# EPICS substitutions: OPCUA/OPCUA-IOC-01App/Db/MAPS_vacuum.substitutions
file "$(TOP)/OPCUA-IOC-01App/Db/MAPS_vacuum_other.template" {
	pattern{ P, R, SUBS, DEBUG, RECORD_TYPE, PV_NAME, NAME_PREFIX, NAME_SUFFIX}

#   General records:
	{ "\$(P)", "\$(R)", "\$(SUBS)", "\$(DEBUG=0)", "stringin", "PE_UNDERRANGE", "\$(NAME_PREFIX)", "Statuses.PE_Underrange_Control" }
    { "\$(P)", "\$(R)", "\$(SUBS)", "\$(DEBUG=0)", "stringin", "UNIT",          "\$(NAME_PREFIX)", "Statuses.Pressure_Unit" }
    { "\$(P)", "\$(R)", "\$(SUBS)", "\$(DEBUG=0)", "stringin", "ERROR",         "\$(NAME_PREFIX)", "Statuses.TPG_Error" }
    { "\$(P)", "\$(R)", "\$(SUBS)", "\$(DEBUG=0)", "bi",       "HEALTHY",       "\$(NAME_PREFIX)", "Statuses.TPG_Healthy" }

#   Channel 1 / Sensor A1:
    { "\$(P)", "\$(R)", "\$(SUBS)", "\$(DEBUG=0)", "stringin", "MEASURED_VALUE_A1",    "\$(NAME_PREFIX)", "Sensor_A1.Measured_Value_Status" }
    { "\$(P)", "\$(R)", "\$(SUBS)", "\$(DEBUG=0)", "stringin", "MEASURING_CIRCUIT_A1", "\$(NAME_PREFIX)", "Sensor_A1.Measuring_Circuit_Status" }
    { "\$(P)", "\$(R)", "\$(SUBS)", "\$(DEBUG=0)", "stringin", "FILTER_TIME_CONST_A1", "\$(NAME_PREFIX)", "Sensor_A1.Filter_Time_Constant" }

#   Relay 1:
    { "\$(P)", "\$(R)", "\$(SUBS)", "\$(DEBUG=0)", "ai",       "THRESHOLD_LOW_A1",      "\$(NAME_PREFIX)", "Relay1.Lower_Threshold" }
    { "\$(P)", "\$(R)", "\$(SUBS)", "\$(DEBUG=0)", "ai",       "THRESHOLD_HI_A1",       "\$(NAME_PREFIX)", "Relay1.Upper_Threshold" }
    { "\$(P)", "\$(R)", "\$(SUBS)", "\$(DEBUG=0)", "stringin", "SWITCH_FUNC_ASSIGN_A1", "\$(NAME_PREFIX)", "Relay1.Switching_Function_Assignment" }
    { "\$(P)", "\$(R)", "\$(SUBS)", "\$(DEBUG=0)", "stringin", "SWITCH_FUNC_STATUS_A1", "\$(NAME_PREFIX)", "Relay1.Switching_Function_Status" }

#   Channel 2 / Sensor A2:
    { "\$(P)", "\$(R)", "\$(SUBS)", "\$(DEBUG=0)", "stringin", "MEASURED_VALUE_A2",    "\$(NAME_PREFIX)", "Sensor_A2.Measured_Value_Status" }
    { "\$(P)", "\$(R)", "\$(SUBS)", "\$(DEBUG=0)", "stringin", "MEASURING_CIRCUIT_A2", "\$(NAME_PREFIX)", "Sensor_A2.Measuring_Circuit_Status" }
    { "\$(P)", "\$(R)", "\$(SUBS)", "\$(DEBUG=0)", "stringin", "FILTER_TIME_CONST_A2", "\$(NAME_PREFIX)", "Sensor_A2.Filter_Time_Constant" }

#   Relay 2:
    { "\$(P)", "\$(R)", "\$(SUBS)", "\$(DEBUG=0)", "ai",       "THRESHOLD_LOW_A2",      "\$(NAME_PREFIX)", "Relay2.Lower_Threshold" }
    { "\$(P)", "\$(R)", "\$(SUBS)", "\$(DEBUG=0)", "ai",       "THRESHOLD_HI_A2",       "\$(NAME_PREFIX)", "Relay2.Upper_Threshold" }
    { "\$(P)", "\$(R)", "\$(SUBS)", "\$(DEBUG=0)", "stringin", "SWITCH_FUNC_ASSIGN_A2", "\$(NAME_PREFIX)", "Relay2.Switching_Function_Assignment" }
    { "\$(P)", "\$(R)", "\$(SUBS)", "\$(DEBUG=0)", "stringin", "SWITCH_FUNC_STATUS_A2", "\$(NAME_PREFIX)", "Relay2.Switching_Function_Status" }

#   Channel 3 / Sensor B1:
    { "\$(P)", "\$(R)", "\$(SUBS)", "\$(DEBUG=0)", "stringin", "MEASURED_VALUE_B1",    "\$(NAME_PREFIX)", "Sensor_B1.Measured_Value_Status" }
    { "\$(P)", "\$(R)", "\$(SUBS)", "\$(DEBUG=0)", "stringin", "MEASURING_CIRCUIT_B1", "\$(NAME_PREFIX)", "Sensor_B1.Measuring_Circuit_Status" }
    { "\$(P)", "\$(R)", "\$(SUBS)", "\$(DEBUG=0)", "stringin", "FILTER_TIME_CONST_B1", "\$(NAME_PREFIX)", "Sensor_B1.Filter_Time_Constant" }

#   Relay 3:
    { "\$(P)", "\$(R)", "\$(SUBS)", "\$(DEBUG=0)", "ai",       "THRESHOLD_LOW_B1",      "\$(NAME_PREFIX)", "Relay3.Lower_Threshold" }
    { "\$(P)", "\$(R)", "\$(SUBS)", "\$(DEBUG=0)", "ai",       "THRESHOLD_HI_B1",       "\$(NAME_PREFIX)", "Relay3.Upper_Threshold" }
    { "\$(P)", "\$(R)", "\$(SUBS)", "\$(DEBUG=0)", "stringin", "SWITCH_FUNC_ASSIGN_B1", "\$(NAME_PREFIX)", "Relay3.Switching_Function_Assignment" }
    { "\$(P)", "\$(R)", "\$(SUBS)", "\$(DEBUG=0)", "stringin", "SWITCH_FUNC_STATUS_B1", "\$(NAME_PREFIX)", "Relay3.Switching_Function_Status" }

#   Channel/Sensor 4:
    { "\$(P)", "\$(R)", "\$(SUBS)", "\$(DEBUG=0)", "stringin", "MEASURED_VALUE_B2",    "\$(NAME_PREFIX)", "Sensor_B2.Measured_Value_Status" }
    { "\$(P)", "\$(R)", "\$(SUBS)", "\$(DEBUG=0)", "stringin", "MEASURING_CIRCUIT_B2", "\$(NAME_PREFIX)", "Sensor_B2.Measuring_Circuit_Status" }
    { "\$(P)", "\$(R)", "\$(SUBS)", "\$(DEBUG=0)", "stringin", "FILTER_TIME_CONST_B2", "\$(NAME_PREFIX)", "Sensor_B2.Filter_Time_Constant" }

#   Relay 4:
    { "\$(P)", "\$(R)", "\$(SUBS)", "\$(DEBUG=0)", "ai",       "THRESHOLD_LOW_B2",      "\$(NAME_PREFIX)", "Relay4.Lower_Threshold" }
    { "\$(P)", "\$(R)", "\$(SUBS)", "\$(DEBUG=0)", "ai",       "THRESHOLD_HI_B2",       "\$(NAME_PREFIX)", "Relay4.Upper_Threshold" }
    { "\$(P)", "\$(R)", "\$(SUBS)", "\$(DEBUG=0)", "stringin", "SWITCH_FUNC_ASSIGN_B2", "\$(NAME_PREFIX)", "Relay4.Switching_Function_Assignment" }
    { "\$(P)", "\$(R)", "\$(SUBS)", "\$(DEBUG=0)", "stringin", "SWITCH_FUNC_STATUS_B2", "\$(NAME_PREFIX)", "Relay4.Switching_Function_Status" }
}

# Pressure PVs additionally require 'PREC' and 'autosave' fields
file "$(TOP)/OPCUA-IOC-01App/Db/MAPS_vacuum_pressures.template" {
	pattern{ P, R, SUBS, DEBUG, RECORD_TYPE, PV_NAME, NAME_PREFIX, NAME_SUFFIX}

#   Channel / Sensor:
    { "\$(P)", "\$(R)", "\$(SUBS)", "\$(DEBUG=0)", "ai",       "PRESSURE_A1",           "\$(NAME_PREFIX)", "Sensor_A1.Pressure" }
    { "\$(P)", "\$(R)", "\$(SUBS)", "\$(DEBUG=0)", "ai",       "PRESSURE_A2",           "\$(NAME_PREFIX)", "Sensor_A2.Pressure" }
    { "\$(P)", "\$(R)", "\$(SUBS)", "\$(DEBUG=0)", "ai",       "PRESSURE_B1",           "\$(NAME_PREFIX)", "Sensor_B1.Pressure" }
    { "\$(P)", "\$(R)", "\$(SUBS)", "\$(DEBUG=0)", "ai",       "PRESSURE_B2",           "\$(NAME_PREFIX)", "Sensor_B2.Pressure" }
}
